FUNCTION SignalmappingOutput

(* ==================================== Digitale Ausgaenge ====================================*)
	
	GVL.mb_Input_Coils[0] := Emitter_Rollenband4m;
	GVL.mb_Input_Coils[3] := StartLED;
	GVL.mb_Input_Coils[4] := StopLED;
	GVL.mb_Input_Coils[5] := ResetLED;
	GVL.mb_Input_Coils[6] := HomeLED;
	GVL.mb_Input_Coils[7] := QuitLED;
	GVL.mb_Input_Coils[9] := Foerderband_Vorwaerts;
	GVL.mb_Input_Coils[10] := Foerderband_Rueckwaerts;
	GVL.mb_Input_Coils[11] := AufzugFoerderbandVorwaerts;
	GVL.mb_Input_Coils[12] := AufzugFoerderbandRueckwaerts;
	GVL.mb_Input_Coils[14] := RBGGabelLinks;
	GVL.mb_Input_Coils[15] := RBGGabelRechts;
	GVL.mb_Input_Coils[17] := RFIDExecuteCommand;
(* ==================================== Analoge Ausgaenge ====================================*)
	GVL.mb_Input_Registers[0] := AufzugSollwert;
	GVL.mb_Input_Registers[1] := RBGSollwertX;
	GVL.mb_Input_Registers[2] := RBGSollwertZ;
	GVL.mb_Input_Registers[3] := RFIDCommand;
	GVL.mb_Input_Registers[4] := RFIDWriteData;
	GVL.mb_Input_Registers[5] := RFIDMemoryIndex;

END_FUNCTION

(* stored: Version 1.1.0.1
   POU SignalmappingOutput: Id {2bdbb390-18c0-4372-a0ff-04e8c4b60455}, SpecialFunc None *)
